// TwinCAT 3 PLC project test_cablelength
// ProgramVersion: 3.1.4022.7
// libraries:
//   LCLS General, * (SLAC)
//   lcls-twincat-motion, * (SLAC)
//   PMPS, * (SLAC - LCLS)
//   Tc2_Standard, * (Beckhoff Automation GmbH)
//   Tc2_System, * (Beckhoff Automation GmbH)
//   Tc2_Utilities, * (Beckhoff Automation GmbH)
//   Tc3_Module, * (Beckhoff Automation GmbH)
// project tree:
//   GVLs/ GVL_Devices.TcGVL
//   / PlcTask.TcTTO
//   POUs/ MAIN.TcPOU
// real-time tasks:
//   TASK PlcTask: cycle T#10ms, priority 20, ADS port 350
// motion (NC):
//   TASK NC-Task 1 SAF: cycle T#2ms, priority 4, ADS port 501
//   TASK NC-Task 1 SVB: cycle T#10ms, priority 8, ADS port 511
//   AXIS CableTestAxis (id 1)
//     Dynamic: AccelerationMaximum=500, DecelerationMaximum=500, Acceleration=47.9998, Deceleration=47.9998, Jerk=460.797, DelayTime=0.008
//     Velo: SlowManual=1, Maximum=5
//     OtherSettings: AllowMotionCmdToSlave=true
//     encoder EncType=29
//       EncPara: ScaleFactorNumerator=0.000390625, Offset=-5990, MaxCount=#xffffffff, ReferenceSystem=1
//         SoftEndMinControl: Enable=true
//         SoftEndMaxControl: Enable=true, Range=25
//         Inc: RefSoftSyncMask=#x0000ffff
//     drive DrvType=24
//       Analog: VeloReferenz=12.5, ScaleFactorActTorque=0.1
//       TimeComp: TaskDelayCycles=1
//     controller CtrType=1
//       CtrPara: PriorControlFactor=1
//         PosDiffControl: Time=0.5
//         Observer: BandWidth=20
// I/O:
//   DEVICE Device 1 (EtherCAT), AmsNetId 172.21.148.78.2.1
//     Term 1 (EK1200) [EK1200-5000 EtherCAT Power supply (2A E-Bus)]
//       Term 2 (EL7047)
//       Term 3 (EL5042) [EL5042 2Ch. BiSS-C Encoder]
//       Term 4 (EL2004)
//       Term 5 (EK1110)
// variable links:
//   (this object) <-> Device 1 (EtherCAT)/Term 1 (EK1200)/Term 2 (EL7047)
//     Drive/Inputs/In/nState1 @bit 3 <-> STM Status/Status/Error
//     Drive/Inputs/In/nState1 @bit 7 <-> STM Status/Status/Motor stall
//     Drive/Inputs/In/nState1 @bit 5 <-> STM Status/Status/Moving negative
//     Drive/Inputs/In/nState1 @bit 4 <-> STM Status/Status/Moving positive
//     Drive/Inputs/In/nState1 @bit 1 <-> STM Status/Status/Ready
//     Drive/Inputs/In/nState1 <-> STM Status/Status/Ready to enable
//     Drive/Inputs/In/nState1 @bit 6 <-> STM Status/Status/Torque reduced
//     Drive/Inputs/In/nState1 @bit 2 <-> STM Status/Status/Warning
//     Drive/Inputs/In/nState2 @bit 3 <-> STM Status/Status/Digital input 1
//     Drive/Inputs/In/nState2 @bit 4 <-> STM Status/Status/Digital input 2
//     Drive/Inputs/In/nState2 @bit 5 <-> STM Status/Status/Sync error
//     Drive/Inputs/In/nState2 @bit 7 <-> STM Status/Status/TxPDO Toggle
//     Drive/Inputs/In/nState4 @bit 1 <-> WcState/InputToggle
//     Drive/Inputs/In/nState4 <-> WcState/WcState
//     Drive/Outputs/Out/nCtrl1 <-> STM Control/Control/Enable
//     Drive/Outputs/Out/nCtrl1 @bit 2 <-> STM Control/Control/Reduce torque
//     Drive/Outputs/Out/nCtrl1 @bit 1 <-> STM Control/Control/Reset
//     Drive/Outputs/Out/nCtrl2 @bit 3 <-> STM Control/Control/Digital output 1
//     Drive/Outputs/Out/nDataOut2[0] <-> STM Velocity/Velocity
//   (this object) <-> Device 1 (EtherCAT)/Term 1 (EK1200)/Term 3 (EL5042)
//     Enc/Inputs/In/nComState @bit 1 <-> WcState/InputToggle
//     Enc/Inputs/In/nComState <-> WcState/WcState
//     Enc/Inputs/In/nDataIn1 <-> FB Inputs Channel 2/Position
//     Enc/Inputs/In/nState1 @bit 12 <-> FB Inputs Channel 2/Status/Diag
//     Enc/Inputs/In/nState1 @bit 1 <-> FB Inputs Channel 2/Status/Error
//     Enc/Inputs/In/nState1 @bit 14 <-> FB Inputs Channel 2/Status/Input cycle counter
//     Enc/Inputs/In/nState1 @bit 2 <-> FB Inputs Channel 2/Status/Ready
//     Enc/Inputs/In/nState1 @bit 13 <-> FB Inputs Channel 2/Status/TxPDO State
//     Enc/Inputs/In/nState1 <-> FB Inputs Channel 2/Status/Warning
//   test_cablelength Instance <-> Device 1 (EtherCAT)/Term 1 (EK1200)/Term 3 (EL5042)
//     PlcTask Inputs/GVL_Devices.M1.nRawEncoderULINT <-> FB Inputs Channel 2/Position
//   test_cablelength Instance <-> NC-Task 1 SAF/Axes/CableTestAxis
//     PlcTask Inputs/GVL_Devices.M1.Axis.NcToPlc <-> Outputs/ToPlc
//     PlcTask Outputs/GVL_Devices.M1.Axis.PlcToNc <-> Inputs/FromPlc
//   test_cablelength Instance <-> test_cablelength/test_cablelength Instance
//     PlcTask Inputs/GVL_Devices.M1.bLimitBackwardEnable <-> PlcTask Outputs/GVL_Devices.bLimitBackward
//     PlcTask Inputs/GVL_Devices.M1.bLimitForwardEnable <-> PlcTask Outputs/GVL_Devices.bLimitForward
//     PlcTask Outputs/GVL_Devices.bLimitBackward <-> PlcTask Inputs/GVL_Devices.M1.bLimitBackwardEnable
//     PlcTask Outputs/GVL_Devices.bLimitForward <-> PlcTask Inputs/GVL_Devices.M1.bLimitForwardEnable

CONFIGURATION test_cablelength
    RESOURCE PLC ON TwinCAT3
        TASK PlcTask(INTERVAL := T#10ms, PRIORITY := 20);
        PROGRAM MAIN WITH PlcTask : MAIN;
    END_RESOURCE
END_CONFIGURATION

// ---- GVLs/GVL_Devices.TcGVL
VAR_GLOBAL
    bLimitForward AT %Q* : BOOL := TRUE;
    bLimitBackward AT %Q* : BOOL := TRUE;

    eStageEnableMode : ENUM_StageEnableMode := ENUM_StageEnableMode.ALWAYS;
    {attribute 'TcLinkTo' := '.bLimitForwardEnable  := TIPC^test_cablelength^test_cablelength Instance^PlcTask Outputs^GVL_Devices.bLimitForward;
                              .bLimitBackwardEnable := TIPC^test_cablelength^test_cablelength Instance^PlcTask Outputs^GVL_Devices.bLimitBackward;
                              .nRawEncoderULINT     := TIIB[Term 3 (EL5042)]^FB Inputs Channel 2^Position'}
    {attribute 'pytmc' := '
        pv: TST:LAB:MMS:01
    '}
    M1: ST_MotionStage := (
        bHardwareEnable := TRUE,
        bPowerSelf := TRUE,
        nEnableMode := eStageEnableMode,
        nHomingMode := ENUM_EpicsHomeCmd.NONE,
        sName := 'TST:LAB:MMS:01');
    (*.bLimitForwardEnable  := TIIB[Term 2 (EL7047)]^STM Status^Status^Digital input 1;
                              .bLimitBackwardEnable := TIIB[Term 2 (EL7047)]^STM Status^Status^Digital input 2;*)

END_VAR

// ---- POUs/MAIN.TcPOU
PROGRAM MAIN
VAR
    fbMotionTstLab: FB_MotionStage;
END_VAR

//Run fb Motion Stage
fbMotionTstLab(stMotionStage:=GVL_Devices.M1);

END_PROGRAM
